FUNCTION_BLOCK FB_Horn
VAR_INPUT
	horn:	E_Horn;
END_VAR
VAR_OUTPUT
		Q:		BOOL;
END_VAR
VAR
	ON_TIME:	TIME := T#500MS;
	IMPULS   :TOF;
    PAUSE    :TOF;

END_VAR

CASE horn OF
	e_horn.off:
		ON_TIME := T#0MS;
	e_horn.short:
		ON_TIME := T#3000MS;
	e_horn.long:
		ON_TIME := T#5000MS;
END_CASE

IMPULS(IN:= NOT PAUSE.Q AND NOT IMPULS.Q, PT:= ON_TIME);
IF horn = e_horn.off THEN
	Q := FALSE;
ELSE
	Q := IMPULS.Q;	
END_IF

END_FUNCTION_BLOCK

(* stored: Version 1.1.0.1, ProductVersion 3.1.4024.9
   POU FB_Horn: Id {30db338a-35ce-4efd-97d8-7974ae10b0f5}, SpecialFunc None *)
